PROGRAM MAIN
VAR
END_VAR

VAR_INPUT
	diOne : bool; 
END_VAR

UC_Measurements();

END_PROGRAM

(* stored: Version 1.1.0.1, ProductVersion 3.1.4020.12
   POU MAIN: Id {792df5c1-e270-4baf-b23d-9e1d1bf8f662}, SpecialFunc None *)
